FUNCTION_BLOCK FB_Color
VAR_INPUT
END_VAR
VAR_OUTPUT
END_VAR
VAR
END_VAR

END_FUNCTION_BLOCK

(* stored: Version 1.1.0.1, ProductVersion 3.1.4024.11
   POU FB_Color: Id {94c17106-1fe3-4f89-8da2-5a9b920caf34}, SpecialFunc None *)
